// TIA Portal V20 export
FUNCTION_BLOCK "FB_ChillerTermotek"   // FB540, SCL
{ S7_Optimized_Access := 'TRUE' }
// stored: AutoNumber false, MemoryReserve 100, SetENOAutomatically false
   VAR
      sTimeHeadChillerHighPressure { S7_SetPoint := 'True'} : TON_TIME;
      sTimeHeadChillerWaterTemperature { S7_SetPoint := 'True'} : TON_TIME;
      sTimeHeadChillerAmbiantTemperature { S7_SetPoint := 'True'} : TON_TIME;
      sTimeOutFlowHeadChiller : TON_TIME;
      sTimeOutLevelHeadChiller { S7_SetPoint := 'True'} : TON_TIME;
      sTimeOutHeadChillerGood : TON_TIME;
      sTimeSourceChillerHighPressure { S7_SetPoint := 'True'} : TON_TIME;
      sTimeSourceChillerWaterTemperature { S7_SetPoint := 'True'} : TON_TIME;
      sTimeSourceChillerAmbiantTemperature { S7_SetPoint := 'True'} : TON_TIME;
      sTimeOutFlowSourceChiller : TON_TIME;
      sTimeOutLevelSourceChiller { S7_SetPoint := 'True'} : TON_TIME;
      sTimeOutSourceChillerGood : TON_TIME;
   END_VAR
   VAR CONSTANT
      TIME_CHILLER_HIGH_PRESSURE : Time := T#8s;
      TIME_CHILLER_WATER_TEMPERATURE : Time := T#8s;
      TIME_CHILLER_AMBIANT_TEMPERATURE : Time := T#8s;
      TIME_OUT_FLOW_CHILLER : Time := T#8S;
      TIME_OUT_LEVEL_CHILLER : Time := T#8S;
      TIME_OUT_CHILLER_GOOD : Time := T#8S;
   END_VAR
BEGIN
   REGION Description header 
       //==================================================================================
       // POSALUX Swiss SA / (C) Copyright 2025
       //----------------------------------------------------------------------------------
       // Title: FB_Chiller_Termotek
       // Comment/Function:
       // Author: Fabien Waldt
       // Engineering: TIA Portal v19
       //----------------------------------------------------------------------------------
       // Change log table:
       // Version  | Date     | Expert in charge | Changes applied
       // ---------|----------|------------------|------------------------------------
       // 00.00.01 | 20250904 | FWA              | First released version
       // ==================================================================================
   END_REGION

   REGION Head Chiller
       REGION Alarm Head Chiller : High Pressure
           #sTimeHeadChillerHighPressure(IN := "DB_PowerOn".sMachineReadySoft AND NOT "DB_DigitalInputs".sHeadChillerHighPressure.sSWStatus,
                                     PT := #TIME_CHILLER_HIGH_PRESSURE,
                                     Q => "LBP_AlarmMsgs".UserA[02].A70UUxx[04]);
       END_REGION

       REGION Alarm Head Chiller : Water Temperature
           #sTimeHeadChillerWaterTemperature(IN := "DB_PowerOn".sMachineReadySoft AND NOT "DB_DigitalInputs".sHeadChillerWaterTemperature.sSWStatus,
                                         PT := #TIME_CHILLER_WATER_TEMPERATURE,
                                         Q => "LBP_AlarmMsgs".UserA[02].A70UUxx[05]);
       END_REGION

       REGION Alarm Head Chiller : Ambiant Temperature
           #sTimeHeadChillerAmbiantTemperature(IN := "DB_PowerOn".sMachineReadySoft AND NOT "DB_DigitalInputs".sHeadChillerAmbiantTemperature.sSWStatus,
                                           PT := #TIME_CHILLER_AMBIANT_TEMPERATURE,
                                           Q => "LBP_AlarmMsgs".UserA[02].A70UUxx[06]);
       END_REGION

       REGION Alarm Head chiller : water flow error
           #sTimeOutFlowHeadChiller(IN := "DB_PowerOn".sMachineReadySoft AND NOT "DB_DigitalInputs".sHeadChillerFlow.sSWStatus,
                                PT := #TIME_OUT_FLOW_CHILLER,
                                Q => "LBP_AlarmMsgs".UserA[2].A70UUxx[0]);
       END_REGION

       REGION Alarm Head chiller : faulty
           #sTimeOutLevelHeadChiller(IN := "DB_PowerOn".sMachineReadySoft AND NOT "DB_DigitalInputs".sHeadChillerCollectivFault.sSWStatus,
                                 PT := #TIME_OUT_LEVEL_CHILLER,
                                 Q => "LBP_AlarmMsgs".UserA[2].A70UUxx[1]);
       END_REGION

       REGION Alarm Head chiller : water level error
           #sTimeOutHeadChillerGood(IN := "DB_PowerOn".sMachineReadySoft AND NOT "DB_DigitalInputs".sHeadChillerWaterLevel.sSWStatus,
                                PT := #TIME_OUT_CHILLER_GOOD,
                                Q => "LBP_AlarmMsgs".UserA[2].A70UUxx[2]);
       END_REGION
   END_REGION

   REGION Source Chiller
       REGION Alarm Source Chiller : High Pressure
           #sTimeSourceChillerHighPressure(IN := "DB_PowerOn".sMachineReadySoft AND NOT "DB_DigitalInputs".sSourceChillerHighPressure.sSWStatus,
                                           PT := #TIME_CHILLER_HIGH_PRESSURE,
                                           Q => "LBP_AlarmMsgs".UserA[02].A70UUxx[10]);
       END_REGION

       REGION Alarm Source Chiller : Water Temperature
          #sTimeSourceChillerWaterTemperature(IN := "DB_PowerOn".sMachineReadySoft AND NOT "DB_DigitalInputs".sSourceChillerWaterTemperature.sSWStatus,
                                              PT := #TIME_CHILLER_WATER_TEMPERATURE,
                                              Q => "LBP_AlarmMsgs".UserA[02].A70UUxx[11]);
       END_REGION

       REGION Alarm Source Chiller : Ambiant Temperature
           #sTimeSourceChillerAmbiantTemperature(IN := "DB_PowerOn".sMachineReadySoft AND NOT "DB_DigitalInputs".sSourceChillerAmbiantTemperature.sSWStatus,
                                                 PT := #TIME_CHILLER_AMBIANT_TEMPERATURE,
                                                 Q => "LBP_AlarmMsgs".UserA[02].A70UUxx[12]);
       END_REGION

       REGION Alarm Source chiller : water flow error
           #sTimeOutFlowSourceChiller(IN := "DB_PowerOn".sMachineReadySoft AND NOT "DB_DigitalInputs".sSourceChillerFlow.sSWStatus,
                                      PT := #TIME_OUT_FLOW_CHILLER,
                                      Q => "LBP_AlarmMsgs".UserA[2].A70UUxx[7]);
       END_REGION

       REGION Alarm Source chiller : faulty
           #sTimeOutLevelSourceChiller(IN := "DB_PowerOn".sMachineReadySoft AND NOT "DB_DigitalInputs".sSourceChillerWaterLevel.sSWStatus,
                                       PT := #TIME_OUT_LEVEL_CHILLER,
                                       Q => "LBP_AlarmMsgs".UserA[2].A70UUxx[8]);
       END_REGION

       REGION Alarm Source chiller : water level error
           #sTimeOutSourceChillerGood(IN := "DB_PowerOn".sMachineReadySoft AND NOT "DB_DigitalInputs".sSourceChillerCollectivFault.sSWStatus,
                                      PT := #TIME_OUT_CHILLER_GOOD,
                                      Q => "LBP_AlarmMsgs".UserA[2].A70UUxx[9]);
       END_REGION
   END_REGION
END_FUNCTION_BLOCK
